{attribute 'qualified_only'}
VAR_GLOBAL
	fbAlarm : FB_TcAlarm;
END_VAR

(* stored: Version 1.1.0.1, ProductVersion 3.1.4024.12
   GVL gAL: Id {6970ad6a-8c2c-4369-9fec-f533d1fb12ad} *)
